TYPE EL2008_EX EXTENDS EL2008 :
STRUCT
	WcState AT %I* : BOOL;
	State AT %I* : UINT;
END_STRUCT
END_TYPE

(* stored: Version 1.1.0.1, ProductVersion 3.1.4026.18
   DUT EL2008_EX: Id {c69dbdbd-f947-49c7-8575-1d4bc4a26e90} *)
